(* PLC project Unnamed, Unknown Unnamed 1 *)
(* stored: creationDateTime 2013-01-29T14:01:00, modificationDateTime 2013-02-26T15:59:13 *)

TYPE LOGLEVEL : (CRITICAL, WARNING, INFO, DEBUG) := INFO;
END_TYPE

FUNCTION_BLOCK LOGGER
  VAR_INPUT
    TRIG : BOOL;
    MSG : STRING;
    LEVEL : LOGLEVEL := INFO;
  END_VAR
  VAR
    TRIG0 : BOOL;
  END_VAR

IF TRIG AND NOT TRIG0 THEN
{{
 extern int LogMessage(uint8_t level, char* buf, uint32_t size);
 LogMessage(GetFbVar(LEVEL),(char*)GetFbVar(MSG, .body),GetFbVar(MSG, .len));
}}
END_IF;
TRIG0:=TRIG;

          
END_FUNCTION_BLOCK
